// Mitsubishi GX Works2 project: 081024   PLC: Q26UDV

// task Task_01 (event TRUE, interval 0, priority 31): POU_01
// task scrubber (event TRUE, interval 0, priority 31): scrubber
// task carrier_4 (event TRUE, interval 0, priority 31): carrier_4
// task bit_moniter (event TRUE, interval 0, priority 31): bit_moniter
// task tranverser (event TRUE, interval 0, priority 31): tranverser
// task Start_cycle (event TRUE, interval 0, priority 31): Start_cycle
// task couter (event TRUE, interval 0, priority 31): couter
// task shower (event TRUE, interval 0, priority 31): shower
// task dryer_cover (event TRUE, interval 0, priority 31): dryer_cover
// task rocking (event TRUE, interval 0, priority 31): rocking
// task carrier_reset (event TRUE, interval 0, priority 31): carrier_reset
// task program_calculate (event TRUE, interval 0, priority 31): program_calculate
// task pump (event TRUE, interval 0, priority 31): pump
// task tower_lamp (event TRUE, interval 0, priority 31): tower_lamp
// task x-lift (event TRUE, interval 0, priority 31): x-lift
// task temp_system (event TRUE, interval 0, priority 31): temp_system
// task data_carry (event TRUE, interval 0, priority 31): data_carry
// task Alarm (event TRUE, interval 0, priority 31): Alarm
// task pro_time (event TRUE, interval 0, priority 31): pro_time
// task unload (event TRUE, interval 0, priority 31): unload
// task data_logger (event TRUE, interval 0, priority 31): data_logger
// task tempLOCK (event TRUE, interval 0, priority 31): tempLOCK
// task QC_pass (event TRUE, interval 0, priority 31): QC_pass
// task barcode_decode (event TRUE, interval 0, priority 31): barcode_decode
// task start_WR (event TRUE, interval 0, priority 31): start_WR
// task data_logger_R (event TRUE, interval 0, priority 31): data_logger_R
// task DBV3 (event TRUE, interval 0, priority 31): DBV3
// task tank_time_A (event TRUE, interval 0, priority 31): tank_time_A
// task send_to_c (event TRUE, interval 0, priority 31): send_to_c
// task receive_c (event TRUE, interval 0, priority 31): receive_c
// task carrier_1 (event TRUE, interval 0, priority 31): carrier_1
// task carrier_2 (event TRUE, interval 0, priority 31): carrier_2
// task carrier_3 (event TRUE, interval 0, priority 31): carrier_3

PROGRAM Alarm
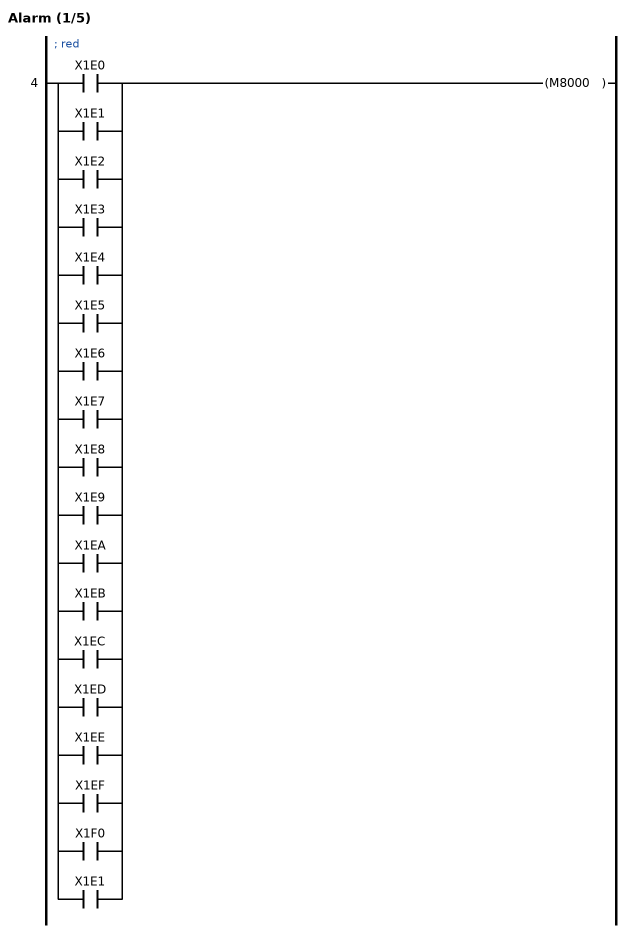
; red
4     LD      X1E0
      OR      X1E1
      OR      X1E2
      OR      X1E3
      OR      X1E4
      OR      X1E5
      OR      X1E6
      OR      X1E7
      OR      X1E8
      OR      X1E9
      OR      X1EA
      OR      X1EB
      OR      X1EC
      OR      X1ED
      OR      X1EE
      OR      X1EF
      OR      X1F0
      OR      X1E1
      OUT     M8000
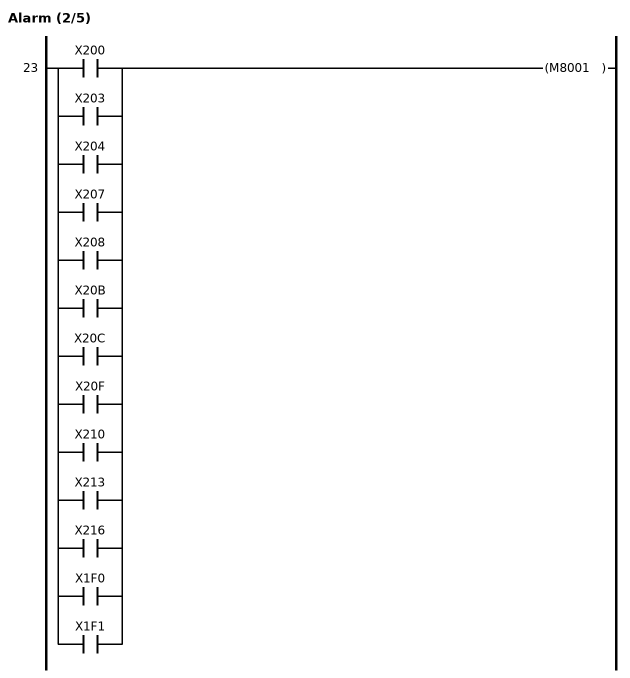
23    LD      X200
      OR      X203
      OR      X204
      OR      X207
      OR      X208
      OR      X20B
      OR      X20C
      OR      X20F
      OR      X210
      OR      X213
      OR      X216
      OR      X1F0
      OR      X1F1
      OUT     M8001
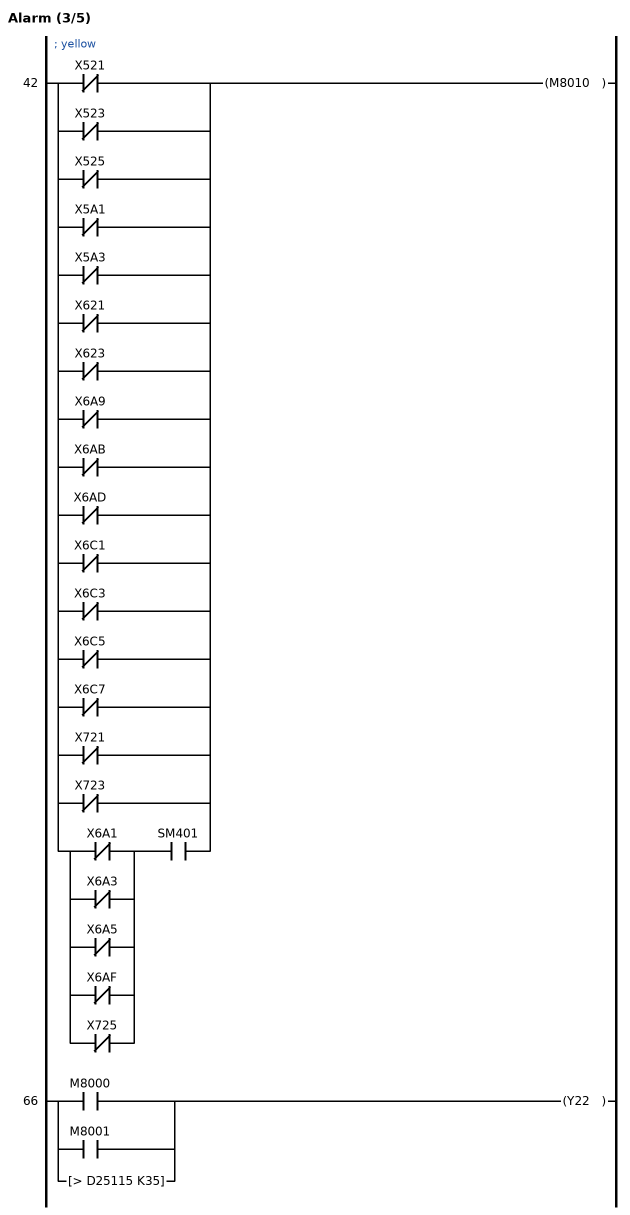
; yellow
42    LDI     X521
      ORI     X523
      ORI     X525
      ORI     X5A1
      ORI     X5A3
      ORI     X621
      ORI     X623
      ORI     X6A9
      ORI     X6AB
      ORI     X6AD
      ORI     X6C1
      ORI     X6C3
      ORI     X6C5
      ORI     X6C7
      ORI     X721
      ORI     X723
      LDI     X6A1
      ORI     X6A3
      ORI     X6A5
      ORI     X6AF
      ORI     X725
      AND     SM401
      ORB
      OUT     M8010
66    LD      M8000
      OR      M8001
      OR>     D25115 K35
      OUT     Y22
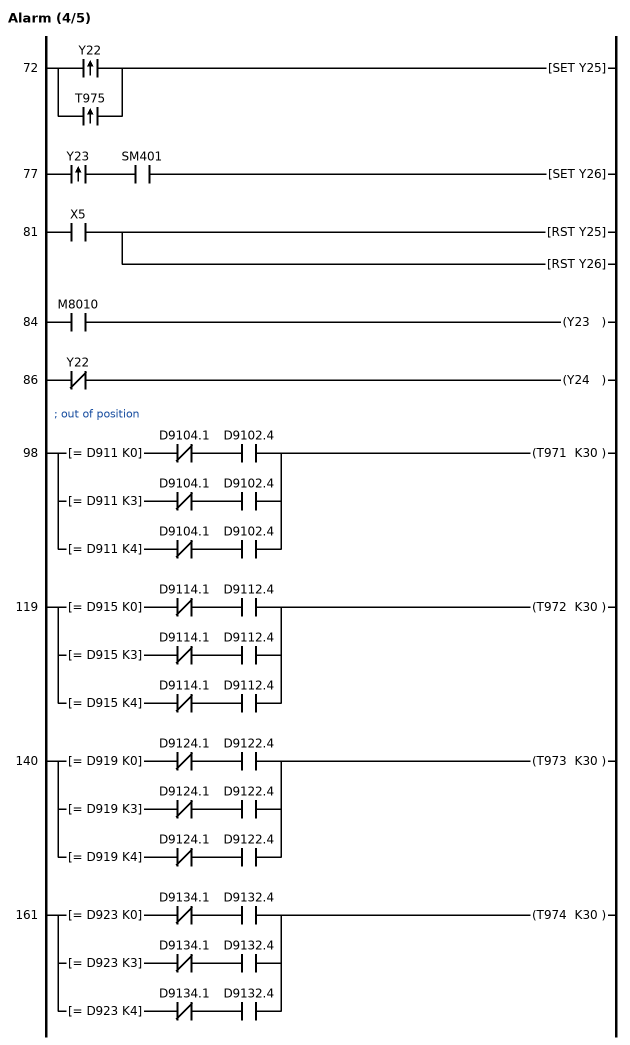
72    LDP     Y22
      ORP     T975
      SET     Y25
77    LDP     Y23
      AND     SM401
      SET     Y26
81    LD      X5
      RST     Y25
      RST     Y26
84    LD      M8010
      OUT     Y23
86    LDI     Y22
      OUT     Y24
; out of position
98    LD=     D911 K0
      ANI     D9104.1
      AND     D9102.4
      LD=     D911 K3
      ANI     D9104.1
      AND     D9102.4
      ORB
      LD=     D911 K4
      ANI     D9104.1
      AND     D9102.4
      ORB
      OUT     T971 K30
119   LD=     D915 K0
      ANI     D9114.1
      AND     D9112.4
      LD=     D915 K3
      ANI     D9114.1
      AND     D9112.4
      ORB
      LD=     D915 K4
      ANI     D9114.1
      AND     D9112.4
      ORB
      OUT     T972 K30
140   LD=     D919 K0
      ANI     D9124.1
      AND     D9122.4
      LD=     D919 K3
      ANI     D9124.1
      AND     D9122.4
      ORB
      LD=     D919 K4
      ANI     D9124.1
      AND     D9122.4
      ORB
      OUT     T973 K30
161   LD=     D923 K0
      ANI     D9134.1
      AND     D9132.4
      LD=     D923 K3
      ANI     D9134.1
      AND     D9132.4
      ORB
      LD=     D923 K4
      ANI     D9134.1
      AND     D9132.4
      ORB
      OUT     T974 K30
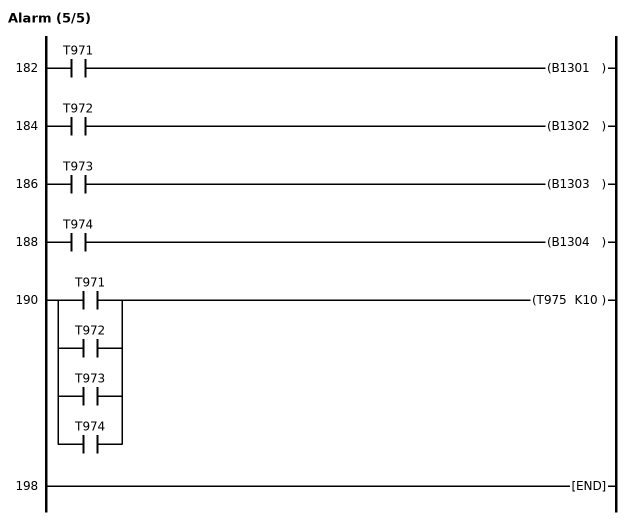
182   LD      T971
      OUT     B1301
184   LD      T972
      OUT     B1302
186   LD      T973
      OUT     B1303
188   LD      T974
      OUT     B1304
190   LD      T971
      OR      T972
      OR      T973
      OR      T974
      OUT     T975 K10
198   END
END_PROGRAM

PROGRAM barcode_decode
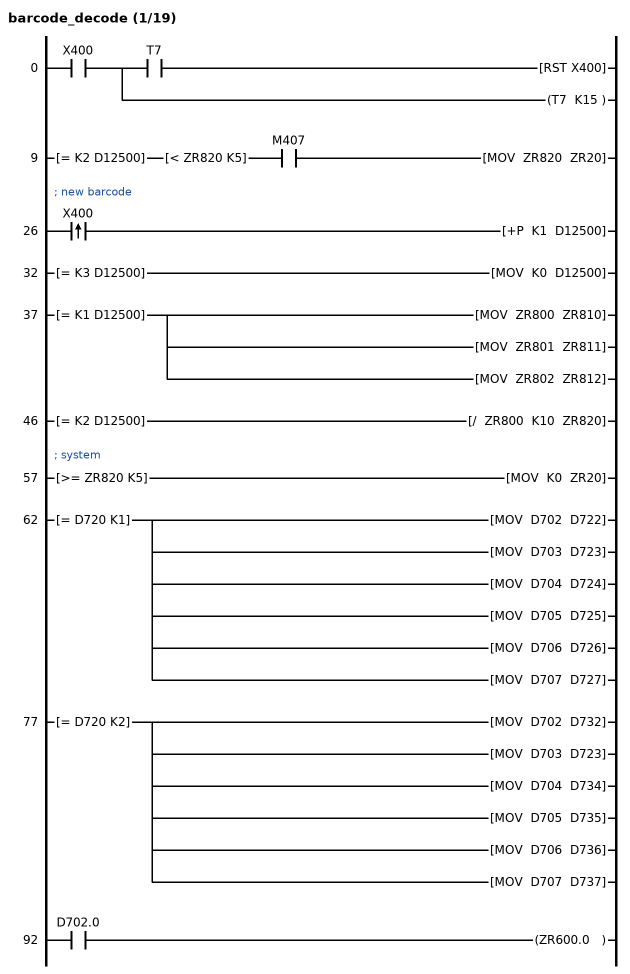
0     LD      X400
      MPS
      AND     T7
      RST     X400
      MPP
      OUT     T7 K15
9     LD=     K2 D12500
      AND<    ZR820 K5
      AND     M407
      MOV     ZR820 ZR20
; new barcode
26    LDP     X400
      +P      K1 D12500
32    LD=     K3 D12500
      MOV     K0 D12500
37    LD=     K1 D12500
      MOV     ZR800 ZR810
      MOV     ZR801 ZR811
      MOV     ZR802 ZR812
46    LD=     K2 D12500
      /       ZR800 K10 ZR820
; system
57    LD>=    ZR820 K5
      MOV     K0 ZR20
62    LD=     D720 K1
      MOV     D702 D722
      MOV     D703 D723
      MOV     D704 D724
      MOV     D705 D725
      MOV     D706 D726
      MOV     D707 D727
77    LD=     D720 K2
      MOV     D702 D732
      MOV     D703 D723
      MOV     D704 D734
      MOV     D705 D735
      MOV     D706 D736
      MOV     D707 D737
92    LD      D702.0
      OUT     ZR600.0
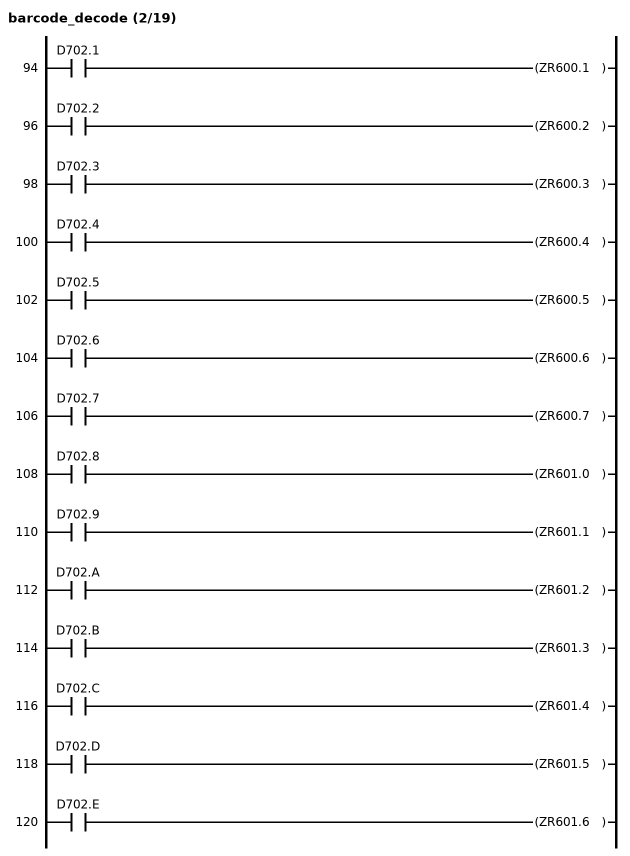
94    LD      D702.1
      OUT     ZR600.1
96    LD      D702.2
      OUT     ZR600.2
98    LD      D702.3
      OUT     ZR600.3
100   LD      D702.4
      OUT     ZR600.4
102   LD      D702.5
      OUT     ZR600.5
104   LD      D702.6
      OUT     ZR600.6
106   LD      D702.7
      OUT     ZR600.7
108   LD      D702.8
      OUT     ZR601.0
110   LD      D702.9
      OUT     ZR601.1
112   LD      D702.A
      OUT     ZR601.2
114   LD      D702.B
      OUT     ZR601.3
116   LD      D702.C
      OUT     ZR601.4
118   LD      D702.D
      OUT     ZR601.5
120   LD      D702.E
      OUT     ZR601.6
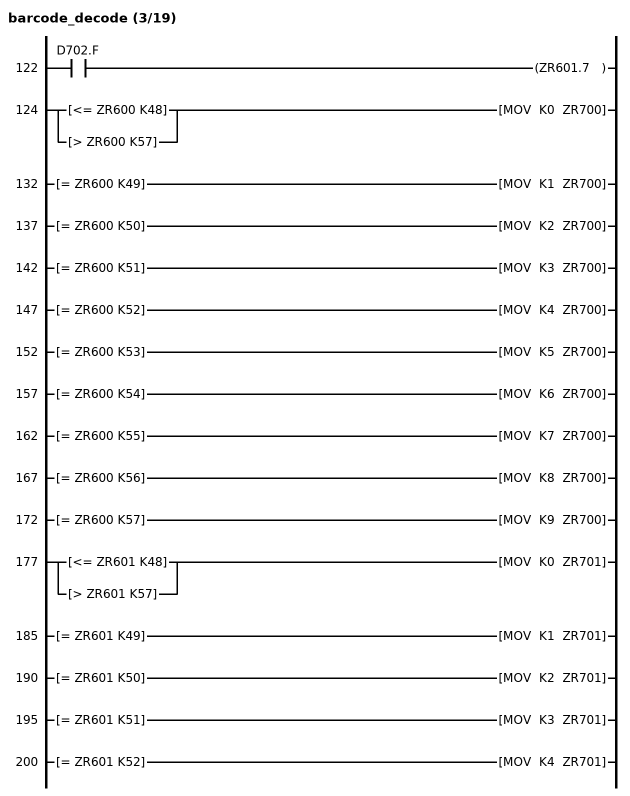
122   LD      D702.F
      OUT     ZR601.7
124   LD<=    ZR600 K48
      OR>     ZR600 K57
      MOV     K0 ZR700
132   LD=     ZR600 K49
      MOV     K1 ZR700
137   LD=     ZR600 K50
      MOV     K2 ZR700
142   LD=     ZR600 K51
      MOV     K3 ZR700
147   LD=     ZR600 K52
      MOV     K4 ZR700
152   LD=     ZR600 K53
      MOV     K5 ZR700
157   LD=     ZR600 K54
      MOV     K6 ZR700
162   LD=     ZR600 K55
      MOV     K7 ZR700
167   LD=     ZR600 K56
      MOV     K8 ZR700
172   LD=     ZR600 K57
      MOV     K9 ZR700
177   LD<=    ZR601 K48
      OR>     ZR601 K57
      MOV     K0 ZR701
185   LD=     ZR601 K49
      MOV     K1 ZR701
190   LD=     ZR601 K50
      MOV     K2 ZR701
195   LD=     ZR601 K51
      MOV     K3 ZR701
200   LD=     ZR601 K52
      MOV     K4 ZR701
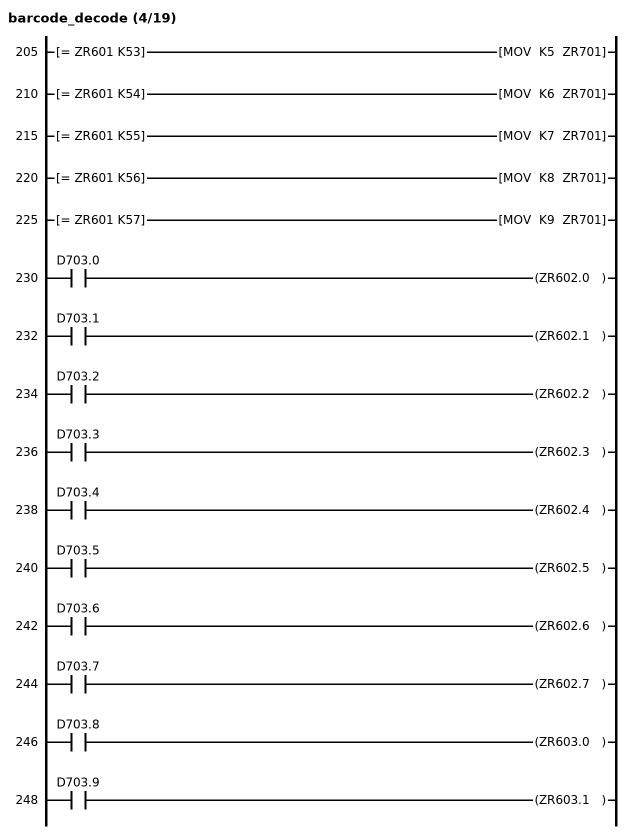
205   LD=     ZR601 K53
      MOV     K5 ZR701
210   LD=     ZR601 K54
      MOV     K6 ZR701
215   LD=     ZR601 K55
      MOV     K7 ZR701
220   LD=     ZR601 K56
      MOV     K8 ZR701
225   LD=     ZR601 K57
      MOV     K9 ZR701
230   LD      D703.0
      OUT     ZR602.0
232   LD      D703.1
      OUT     ZR602.1
234   LD      D703.2
      OUT     ZR602.2
236   LD      D703.3
      OUT     ZR602.3
238   LD      D703.4
      OUT     ZR602.4
240   LD      D703.5
      OUT     ZR602.5
242   LD      D703.6
      OUT     ZR602.6
244   LD      D703.7
      OUT     ZR602.7
246   LD      D703.8
      OUT     ZR603.0
248   LD      D703.9
      OUT     ZR603.1
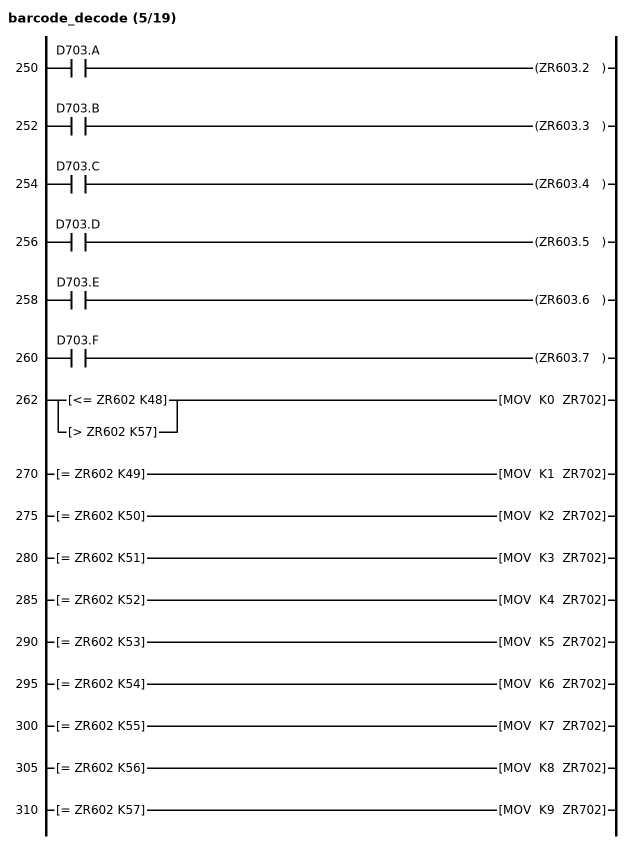
250   LD      D703.A
      OUT     ZR603.2
252   LD      D703.B
      OUT     ZR603.3
254   LD      D703.C
      OUT     ZR603.4
256   LD      D703.D
      OUT     ZR603.5
258   LD      D703.E
      OUT     ZR603.6
260   LD      D703.F
      OUT     ZR603.7
262   LD<=    ZR602 K48
      OR>     ZR602 K57
      MOV     K0 ZR702
270   LD=     ZR602 K49
      MOV     K1 ZR702
275   LD=     ZR602 K50
      MOV     K2 ZR702
280   LD=     ZR602 K51
      MOV     K3 ZR702
285   LD=     ZR602 K52
      MOV     K4 ZR702
290   LD=     ZR602 K53
      MOV     K5 ZR702
295   LD=     ZR602 K54
      MOV     K6 ZR702
300   LD=     ZR602 K55
      MOV     K7 ZR702
305   LD=     ZR602 K56
      MOV     K8 ZR702
310   LD=     ZR602 K57
      MOV     K9 ZR702
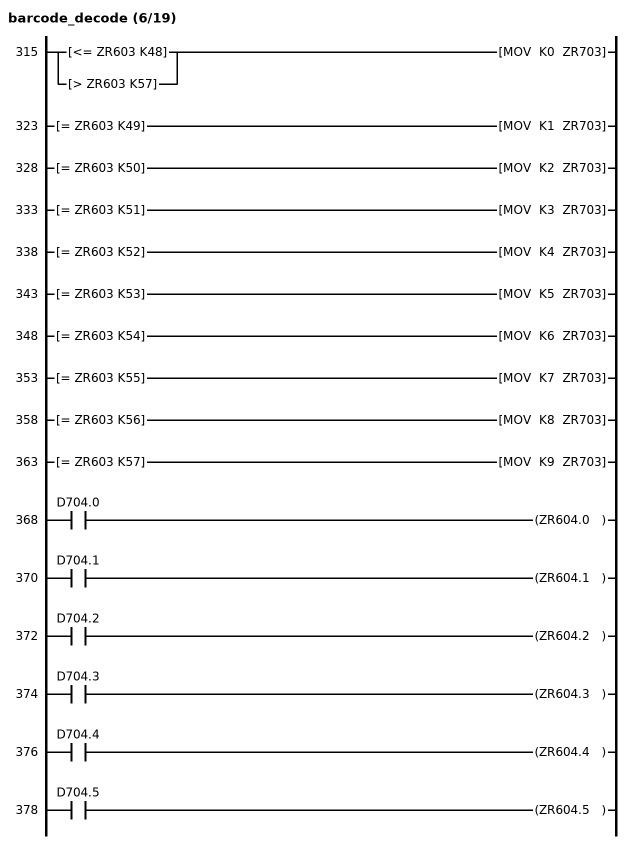
315   LD<=    ZR603 K48
      OR>     ZR603 K57
      MOV     K0 ZR703
323   LD=     ZR603 K49
      MOV     K1 ZR703
328   LD=     ZR603 K50
      MOV     K2 ZR703
333   LD=     ZR603 K51
      MOV     K3 ZR703
338   LD=     ZR603 K52
      MOV     K4 ZR703
343   LD=     ZR603 K53
      MOV     K5 ZR703
348   LD=     ZR603 K54
      MOV     K6 ZR703
353   LD=     ZR603 K55
      MOV     K7 ZR703
358   LD=     ZR603 K56
      MOV     K8 ZR703
363   LD=     ZR603 K57
      MOV     K9 ZR703
368   LD      D704.0
      OUT     ZR604.0
370   LD      D704.1
      OUT     ZR604.1
372   LD      D704.2
      OUT     ZR604.2
374   LD      D704.3
      OUT     ZR604.3
376   LD      D704.4
      OUT     ZR604.4
378   LD      D704.5
      OUT     ZR604.5
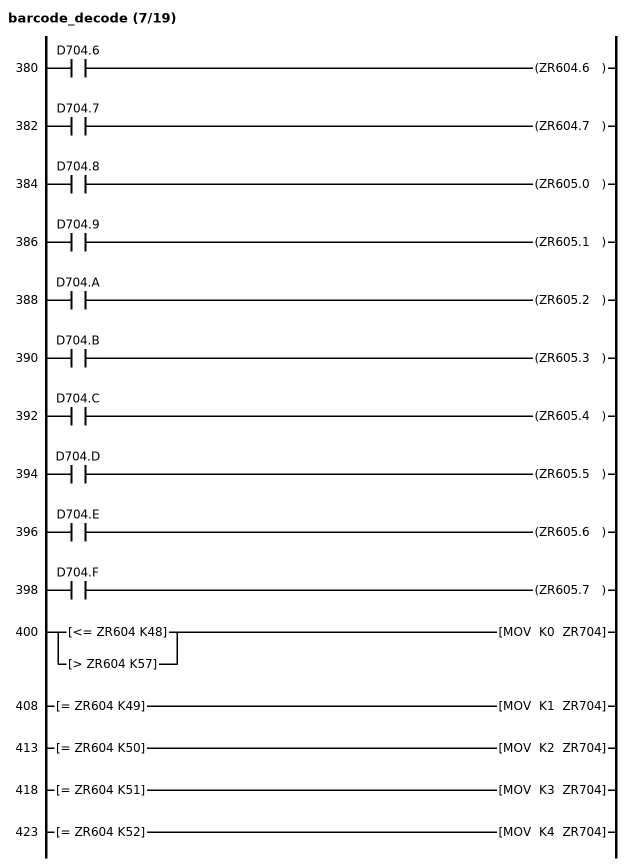
380   LD      D704.6
      OUT     ZR604.6
382   LD      D704.7
      OUT     ZR604.7
384   LD      D704.8
      OUT     ZR605.0
386   LD      D704.9
      OUT     ZR605.1
388   LD      D704.A
      OUT     ZR605.2
390   LD      D704.B
      OUT     ZR605.3
392   LD      D704.C
      OUT     ZR605.4
394   LD      D704.D
      OUT     ZR605.5
396   LD      D704.E
      OUT     ZR605.6
398   LD      D704.F
      OUT     ZR605.7
400   LD<=    ZR604 K48
      OR>     ZR604 K57
      MOV     K0 ZR704
408   LD=     ZR604 K49
      MOV     K1 ZR704
413   LD=     ZR604 K50
      MOV     K2 ZR704
418   LD=     ZR604 K51
      MOV     K3 ZR704
423   LD=     ZR604 K52
      MOV     K4 ZR704
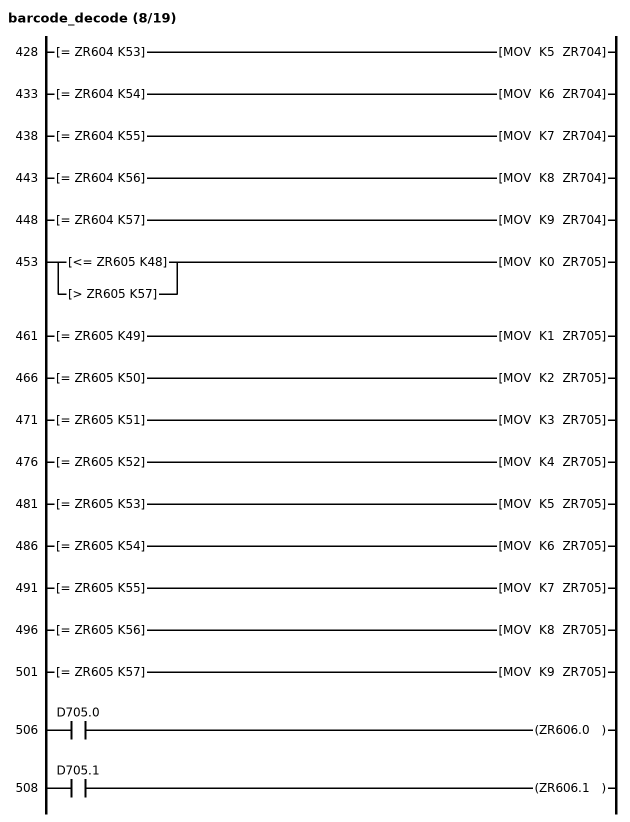
428   LD=     ZR604 K53
      MOV     K5 ZR704
433   LD=     ZR604 K54
      MOV     K6 ZR704
438   LD=     ZR604 K55
      MOV     K7 ZR704
443   LD=     ZR604 K56
      MOV     K8 ZR704
448   LD=     ZR604 K57
      MOV     K9 ZR704
453   LD<=    ZR605 K48
      OR>     ZR605 K57
      MOV     K0 ZR705
461   LD=     ZR605 K49
      MOV     K1 ZR705
466   LD=     ZR605 K50
      MOV     K2 ZR705
471   LD=     ZR605 K51
      MOV     K3 ZR705
476   LD=     ZR605 K52
      MOV     K4 ZR705
481   LD=     ZR605 K53
      MOV     K5 ZR705
486   LD=     ZR605 K54
      MOV     K6 ZR705
491   LD=     ZR605 K55
      MOV     K7 ZR705
496   LD=     ZR605 K56
      MOV     K8 ZR705
501   LD=     ZR605 K57
      MOV     K9 ZR705
506   LD      D705.0
      OUT     ZR606.0
508   LD      D705.1
      OUT     ZR606.1
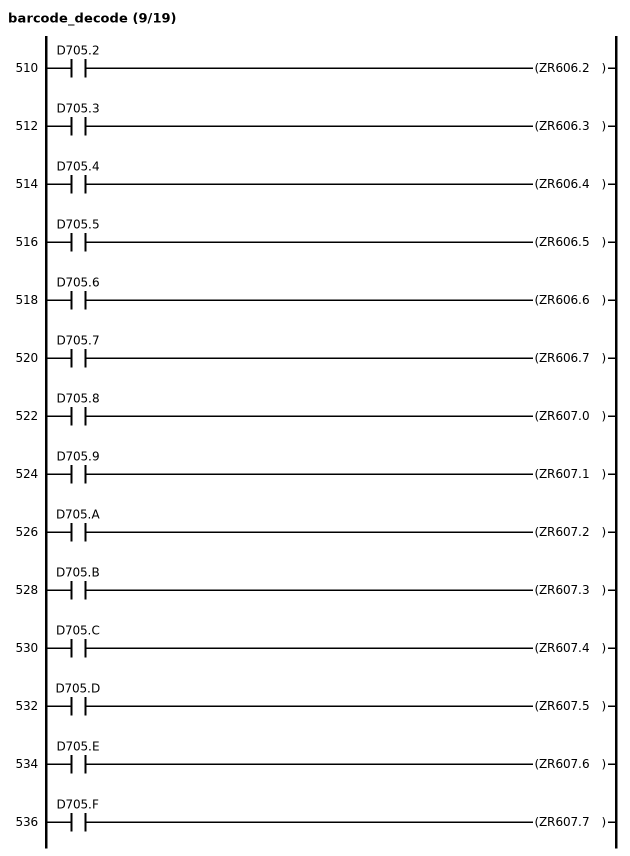
510   LD      D705.2
      OUT     ZR606.2
512   LD      D705.3
      OUT     ZR606.3
514   LD      D705.4
      OUT     ZR606.4
516   LD      D705.5
      OUT     ZR606.5
518   LD      D705.6
      OUT     ZR606.6
520   LD      D705.7
      OUT     ZR606.7
522   LD      D705.8
      OUT     ZR607.0
524   LD      D705.9
      OUT     ZR607.1
526   LD      D705.A
      OUT     ZR607.2
528   LD      D705.B
      OUT     ZR607.3
530   LD      D705.C
      OUT     ZR607.4
532   LD      D705.D
      OUT     ZR607.5
534   LD      D705.E
      OUT     ZR607.6
536   LD      D705.F
      OUT     ZR607.7
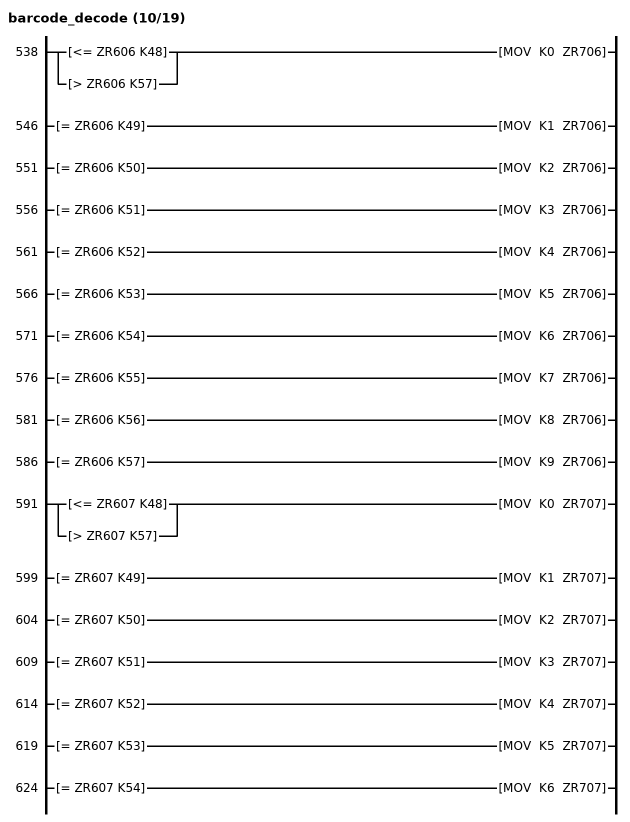
538   LD<=    ZR606 K48
      OR>     ZR606 K57
      MOV     K0 ZR706
546   LD=     ZR606 K49
      MOV     K1 ZR706
551   LD=     ZR606 K50
      MOV     K2 ZR706
556   LD=     ZR606 K51
      MOV     K3 ZR706
561   LD=     ZR606 K52
      MOV     K4 ZR706
566   LD=     ZR606 K53
      MOV     K5 ZR706
571   LD=     ZR606 K54
      MOV     K6 ZR706
576   LD=     ZR606 K55
      MOV     K7 ZR706
581   LD=     ZR606 K56
      MOV     K8 ZR706
586   LD=     ZR606 K57
      MOV     K9 ZR706
591   LD<=    ZR607 K48
      OR>     ZR607 K57
      MOV     K0 ZR707
599   LD=     ZR607 K49
      MOV     K1 ZR707
604   LD=     ZR607 K50
      MOV     K2 ZR707
609   LD=     ZR607 K51
      MOV     K3 ZR707
614   LD=     ZR607 K52
      MOV     K4 ZR707
619   LD=     ZR607 K53
      MOV     K5 ZR707
624   LD=     ZR607 K54
      MOV     K6 ZR707
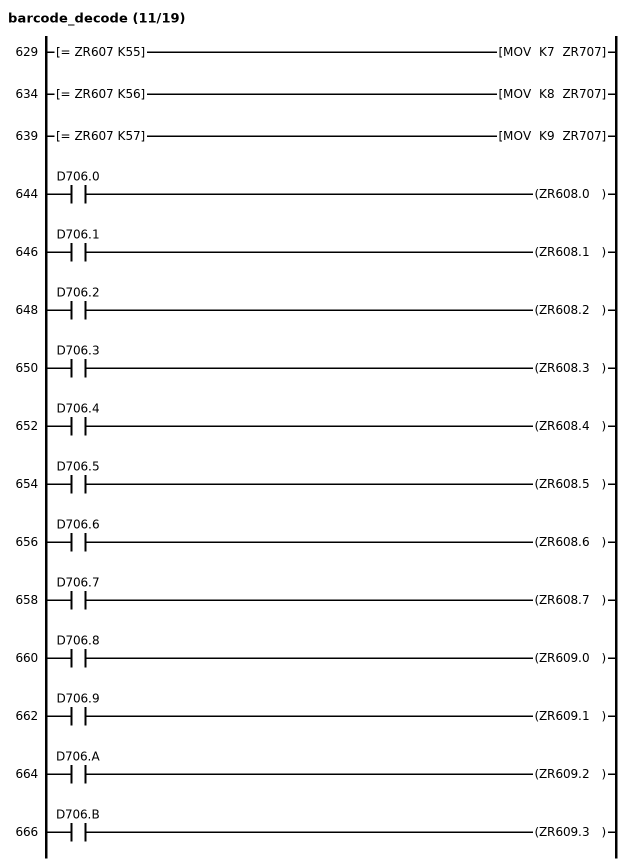
629   LD=     ZR607 K55
      MOV     K7 ZR707
634   LD=     ZR607 K56
      MOV     K8 ZR707
639   LD=     ZR607 K57
      MOV     K9 ZR707
644   LD      D706.0
      OUT     ZR608.0
646   LD      D706.1
      OUT     ZR608.1
648   LD      D706.2
      OUT     ZR608.2
650   LD      D706.3
      OUT     ZR608.3
652   LD      D706.4
      OUT     ZR608.4
654   LD      D706.5
      OUT     ZR608.5
656   LD      D706.6
      OUT     ZR608.6
658   LD      D706.7
      OUT     ZR608.7
660   LD      D706.8
      OUT     ZR609.0
662   LD      D706.9
      OUT     ZR609.1
664   LD      D706.A
      OUT     ZR609.2
666   LD      D706.B
      OUT     ZR609.3
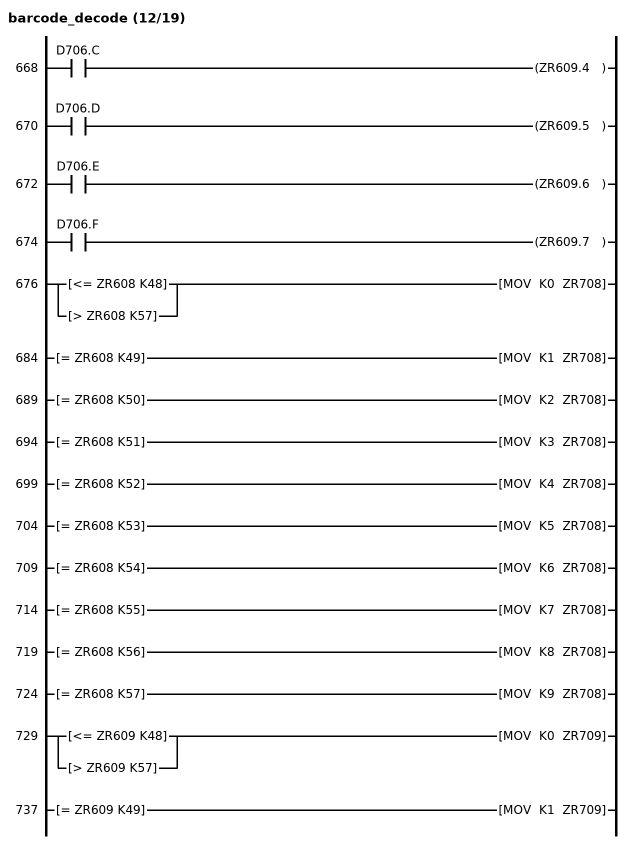
668   LD      D706.C
      OUT     ZR609.4
670   LD      D706.D
      OUT     ZR609.5
672   LD      D706.E
      OUT     ZR609.6
674   LD      D706.F
      OUT     ZR609.7
676   LD<=    ZR608 K48
      OR>     ZR608 K57
      MOV     K0 ZR708
684   LD=     ZR608 K49
      MOV     K1 ZR708
689   LD=     ZR608 K50
      MOV     K2 ZR708
694   LD=     ZR608 K51
      MOV     K3 ZR708
699   LD=     ZR608 K52
      MOV     K4 ZR708
704   LD=     ZR608 K53
      MOV     K5 ZR708
709   LD=     ZR608 K54
      MOV     K6 ZR708
714   LD=     ZR608 K55
      MOV     K7 ZR708
719   LD=     ZR608 K56
      MOV     K8 ZR708
724   LD=     ZR608 K57
      MOV     K9 ZR708
729   LD<=    ZR609 K48
      OR>     ZR609 K57
      MOV     K0 ZR709
737   LD=     ZR609 K49
      MOV     K1 ZR709
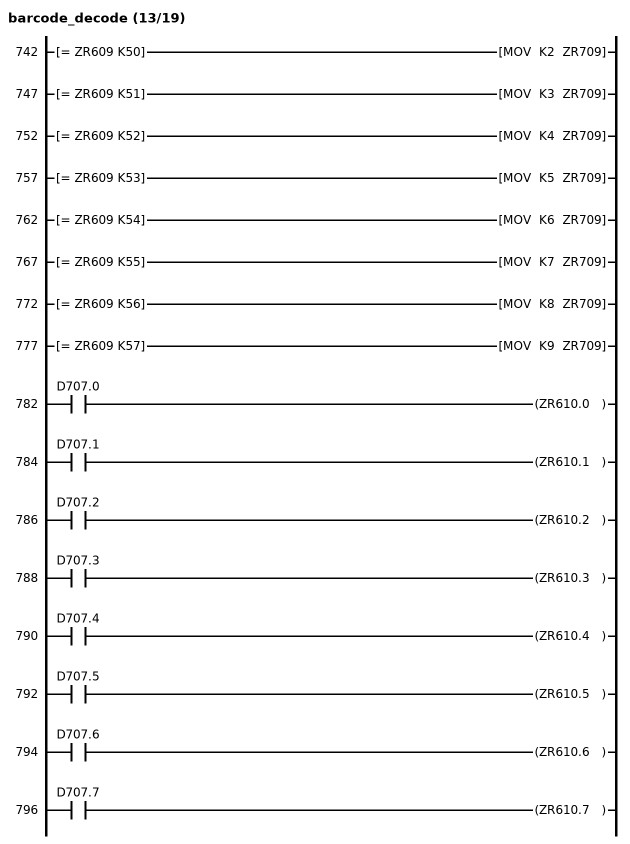
742   LD=     ZR609 K50
      MOV     K2 ZR709
747   LD=     ZR609 K51
      MOV     K3 ZR709
752   LD=     ZR609 K52
      MOV     K4 ZR709
757   LD=     ZR609 K53
      MOV     K5 ZR709
762   LD=     ZR609 K54
      MOV     K6 ZR709
767   LD=     ZR609 K55
      MOV     K7 ZR709
772   LD=     ZR609 K56
      MOV     K8 ZR709
777   LD=     ZR609 K57
      MOV     K9 ZR709
782   LD      D707.0
      OUT     ZR610.0
784   LD      D707.1
      OUT     ZR610.1
786   LD      D707.2
      OUT     ZR610.2
788   LD      D707.3
      OUT     ZR610.3
790   LD      D707.4
      OUT     ZR610.4
792   LD      D707.5
      OUT     ZR610.5
794   LD      D707.6
      OUT     ZR610.6
796   LD      D707.7
      OUT     ZR610.7
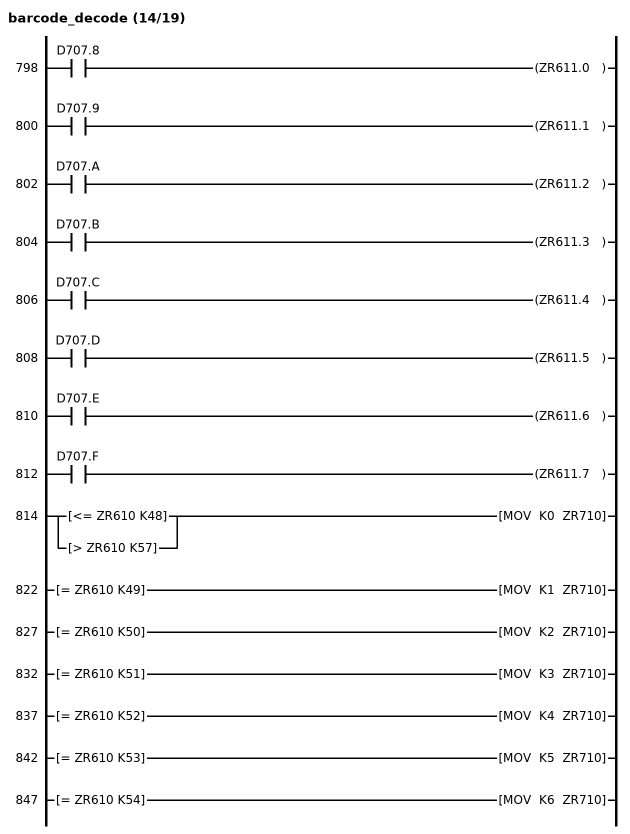
798   LD      D707.8
      OUT     ZR611.0
800   LD      D707.9
      OUT     ZR611.1
802   LD      D707.A
      OUT     ZR611.2
804   LD      D707.B
      OUT     ZR611.3
806   LD      D707.C
      OUT     ZR611.4
808   LD      D707.D
      OUT     ZR611.5
810   LD      D707.E
      OUT     ZR611.6
812   LD      D707.F
      OUT     ZR611.7
814   LD<=    ZR610 K48
      OR>     ZR610 K57
      MOV     K0 ZR710
822   LD=     ZR610 K49
      MOV     K1 ZR710
827   LD=     ZR610 K50
      MOV     K2 ZR710
832   LD=     ZR610 K51
      MOV     K3 ZR710
837   LD=     ZR610 K52
      MOV     K4 ZR710
842   LD=     ZR610 K53
      MOV     K5 ZR710
847   LD=     ZR610 K54
      MOV     K6 ZR710
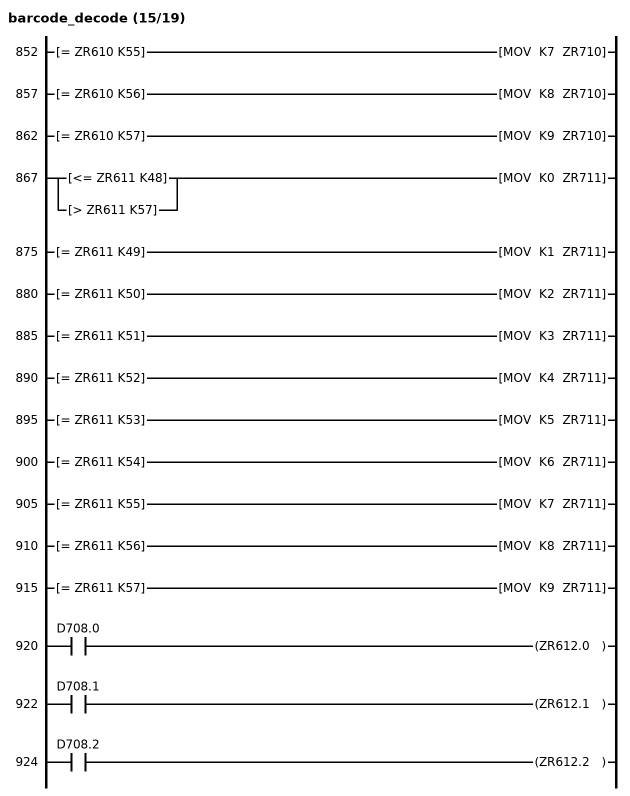
852   LD=     ZR610 K55
      MOV     K7 ZR710
857   LD=     ZR610 K56
      MOV     K8 ZR710
862   LD=     ZR610 K57
      MOV     K9 ZR710
867   LD<=    ZR611 K48
      OR>     ZR611 K57
      MOV     K0 ZR711
875   LD=     ZR611 K49
      MOV     K1 ZR711
880   LD=     ZR611 K50
      MOV     K2 ZR711
885   LD=     ZR611 K51
      MOV     K3 ZR711
890   LD=     ZR611 K52
      MOV     K4 ZR711
895   LD=     ZR611 K53
      MOV     K5 ZR711
900   LD=     ZR611 K54
      MOV     K6 ZR711
905   LD=     ZR611 K55
      MOV     K7 ZR711
910   LD=     ZR611 K56
      MOV     K8 ZR711
915   LD=     ZR611 K57
      MOV     K9 ZR711
920   LD      D708.0
      OUT     ZR612.0
922   LD      D708.1
      OUT     ZR612.1
924   LD      D708.2
      OUT     ZR612.2
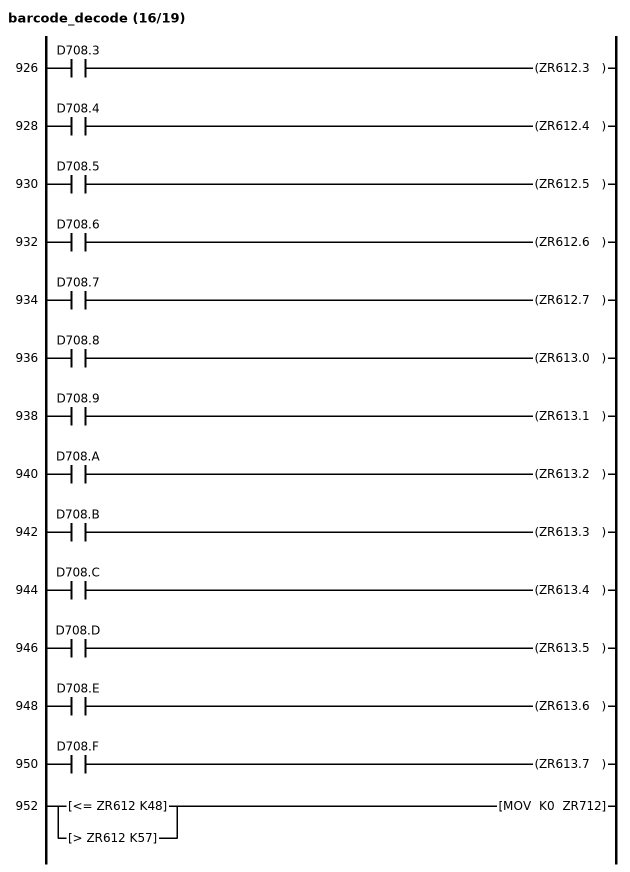
926   LD      D708.3
      OUT     ZR612.3
928   LD      D708.4
      OUT     ZR612.4
930   LD      D708.5
      OUT     ZR612.5
932   LD      D708.6
      OUT     ZR612.6
934   LD      D708.7
      OUT     ZR612.7
936   LD      D708.8
      OUT     ZR613.0
938   LD      D708.9
      OUT     ZR613.1
940   LD      D708.A
      OUT     ZR613.2
942   LD      D708.B
      OUT     ZR613.3
944   LD      D708.C
      OUT     ZR613.4
946   LD      D708.D
      OUT     ZR613.5
948   LD      D708.E
      OUT     ZR613.6
950   LD      D708.F
      OUT     ZR613.7
952   LD<=    ZR612 K48
      OR>     ZR612 K57
      MOV     K0 ZR712
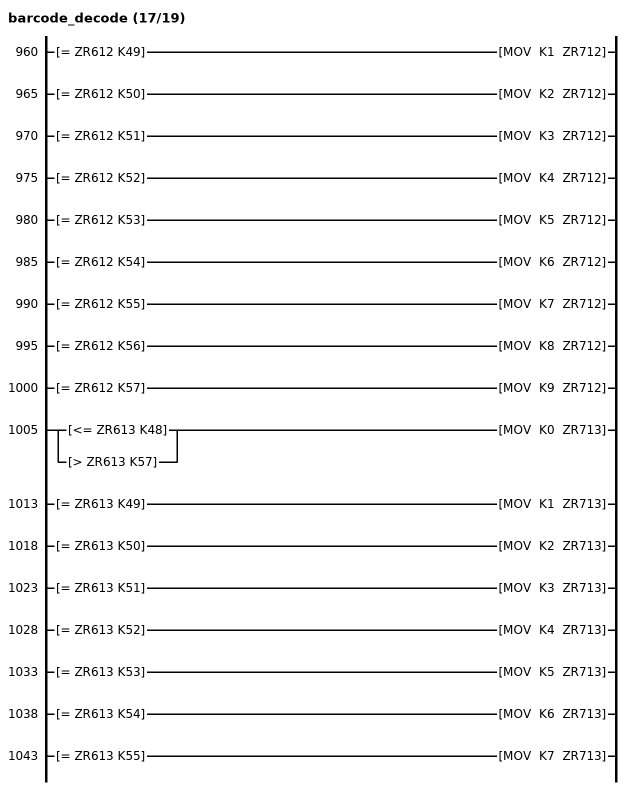
960   LD=     ZR612 K49
      MOV     K1 ZR712
965   LD=     ZR612 K50
      MOV     K2 ZR712
970   LD=     ZR612 K51
      MOV     K3 ZR712
975   LD=     ZR612 K52
      MOV     K4 ZR712
980   LD=     ZR612 K53
      MOV     K5 ZR712
985   LD=     ZR612 K54
      MOV     K6 ZR712
990   LD=     ZR612 K55
      MOV     K7 ZR712
995   LD=     ZR612 K56
      MOV     K8 ZR712
1000  LD=     ZR612 K57
      MOV     K9 ZR712
1005  LD<=    ZR613 K48
      OR>     ZR613 K57
      MOV     K0 ZR713
1013  LD=     ZR613 K49
      MOV     K1 ZR713
1018  LD=     ZR613 K50
      MOV     K2 ZR713
1023  LD=     ZR613 K51
      MOV     K3 ZR713
1028  LD=     ZR613 K52
      MOV     K4 ZR713
1033  LD=     ZR613 K53
      MOV     K5 ZR713
1038  LD=     ZR613 K54
      MOV     K6 ZR713
1043  LD=     ZR613 K55
      MOV     K7 ZR713
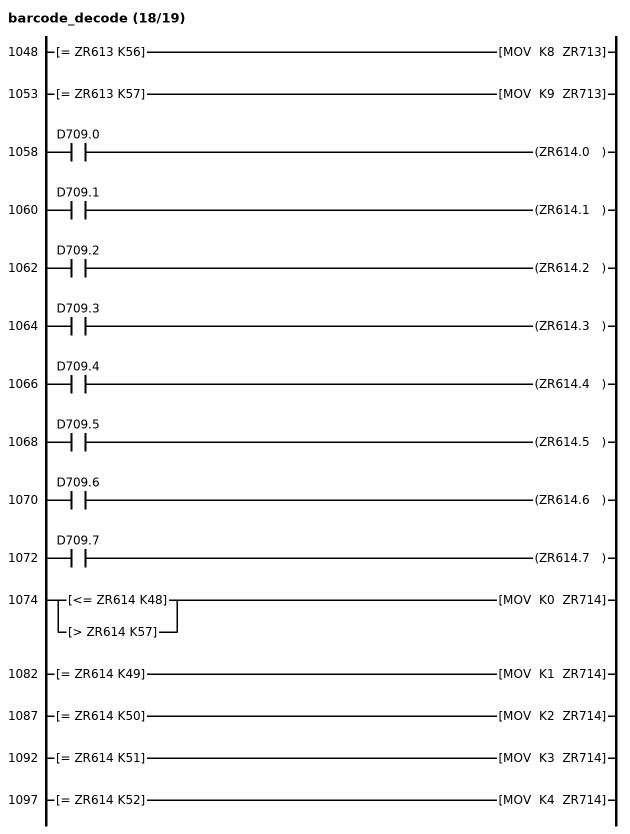
1048  LD=     ZR613 K56
      MOV     K8 ZR713
1053  LD=     ZR613 K57
      MOV     K9 ZR713
1058  LD      D709.0
      OUT     ZR614.0
1060  LD      D709.1
      OUT     ZR614.1
1062  LD      D709.2
      OUT     ZR614.2
1064  LD      D709.3
      OUT     ZR614.3
1066  LD      D709.4
      OUT     ZR614.4
1068  LD      D709.5
      OUT     ZR614.5
1070  LD      D709.6
      OUT     ZR614.6
1072  LD      D709.7
      OUT     ZR614.7
1074  LD<=    ZR614 K48
      OR>     ZR614 K57
      MOV     K0 ZR714
1082  LD=     ZR614 K49
      MOV     K1 ZR714
1087  LD=     ZR614 K50
      MOV     K2 ZR714
1092  LD=     ZR614 K51
      MOV     K3 ZR714
1097  LD=     ZR614 K52
      MOV     K4 ZR714
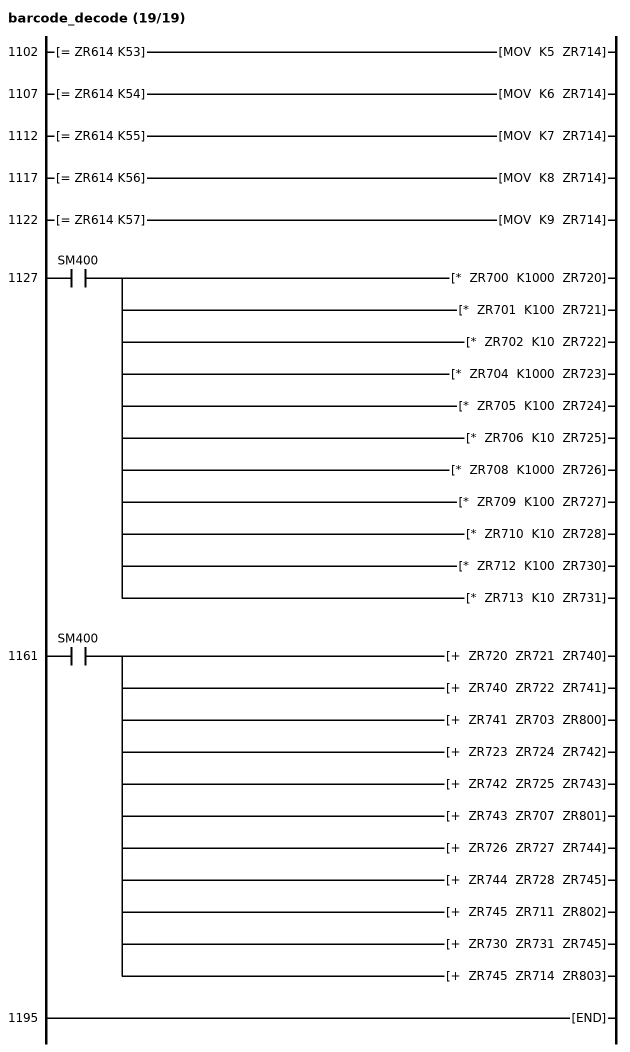
1102  LD=     ZR614 K53
      MOV     K5 ZR714
1107  LD=     ZR614 K54
      MOV     K6 ZR714
1112  LD=     ZR614 K55
      MOV     K7 ZR714
1117  LD=     ZR614 K56
      MOV     K8 ZR714
1122  LD=     ZR614 K57
      MOV     K9 ZR714
1127  LD      SM400
      *       ZR700 K1000 ZR720
      *       ZR701 K100 ZR721
      *       ZR702 K10 ZR722
      *       ZR704 K1000 ZR723
      *       ZR705 K100 ZR724
      *       ZR706 K10 ZR725
      *       ZR708 K1000 ZR726
      *       ZR709 K100 ZR727
      *       ZR710 K10 ZR728
      *       ZR712 K100 ZR730
      *       ZR713 K10 ZR731
1161  LD      SM400
      +       ZR720 ZR721 ZR740
      +       ZR740 ZR722 ZR741
      +       ZR741 ZR703 ZR800
      +       ZR723 ZR724 ZR742
      +       ZR742 ZR725 ZR743
      +       ZR743 ZR707 ZR801
      +       ZR726 ZR727 ZR744
      +       ZR744 ZR728 ZR745
      +       ZR745 ZR711 ZR802
      +       ZR730 ZR731 ZR745
      +       ZR745 ZR714 ZR803
1195  END
END_PROGRAM

PROGRAM bit_moniter
